FUNCTION_BLOCK FB_ComponentBase_SR EXTENDS FB_ComponentBase
VAR_INPUT
END_VAR

VAR_OUTPUT
END_VAR

VAR
    Comp_Alarms : ARRAY[1..20] OF FB_TcAlarm;

    i : UDINT;

END_VAR

METHOD ClearAlarms
VAR_INPUT
    MyAlarms : ARRAY[1..Global.MAX_ALARM_COUNT] OF FB_TcAlarm;
END_VAR

VAR
    i : UDINT;
END_VAR
FOR i := 1 TO Global.MAX_ALARM_COUNT DO
    MyAlarms[i].Clear(0, 0);
END_FOR;
END_METHOD

METHOD RaiseAlarm2Args
VAR_IN_OUT
    fbAlarm : FB_TcAlarm; //Alarm to be raised
END_VAR

VAR_INPUT
    String_1 : STRING; //First String Parameter (The Name of this component will be applied first automatically)
    String_2 : STRING; //Second String Parameter
END_VAR
F_RaiseAlarmWithStringParameters(Alarm := fbAlarm, String_1 := Name, String_2 := String_1, String_3 := String_2);
END_METHOD

METHOD Reset : BOOL
_Error   := FALSE;
_ErrorID := 0;

IF SUPER^.Reset() THEN
    Reset := TRUE;
END_IF
END_METHOD

END_FUNCTION_BLOCK

(* stored: Version 1.1.0.1
   POU FB_ComponentBase_SR: Id {ff7dc399-0fd3-4f30-ad77-8c6bfec79dda}, SpecialFunc None
   Folder Methods: Id {7b22317b-ca0d-4a05-9f65-ebb790dfcf5a}
   Folder Properties: Id {0429b360-a469-401b-a985-cdad475e14e7}
   Method ClearAlarms: Id {e576e51a-e7ca-435e-8632-a9e461cc0f08}
   Method RaiseAlarm2Args: Id {89d22782-64bd-4c9b-9078-27d9d028765d}
   Method Reset: Id {5350edae-f92c-4067-941d-83a15372d499} *)
